RoboDK station: kr10 camera 070819 First 4 poses.rdk

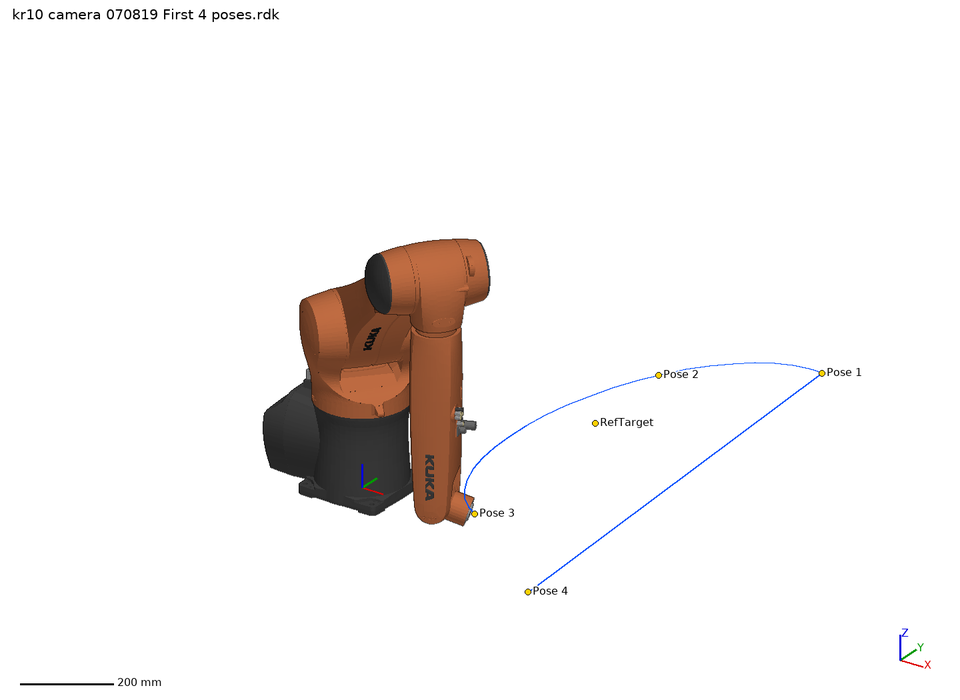
[picture v0: the station drawn from its stored meshes, robots at their saved joint values, targets as dots, program paths as lines]
Station kr10 camera 070819 First 4 poses. Poses are relative to the parent item; angles as X-Y-Z fixed-axis rotations.
  - frame KUKA KR 10 R1100 sixx Base at (0, 0, 0) mm
    - robot KUKA KR 10 R1100 sixx: 6 axes, payload 10 kg, reach 1101 mm, repeatability 0.03 mm, weight 54 kg
        modified DH rows (alpha deg, a mm, theta deg, d mm): 0, 0, 0, 400; -90, 25, 0, 0; 0, 560, -90, 0; -90, 35, 0, 515; 90, 0, 0, 0; -90, 0, 180, 80
        joint limits [-170, -190, -120, -185, -120, -350] to [170, 45, 156, 185, 120, 350]; home [0, -90, 90, 0, 0, 0]; saved at [37.108, -35.584, 126.083, 60.338, -72.571, -20.944]
      - tool Tool 1, TCP at (0, 0, 10) mm
    - target RefTarget (Cartesian target) at (609.71, 0, 323.9) mm, rotated rx 0 ry 90 rz 0 deg; joints [0, -49.182, 128.637, 0, -79.455, 0] of KUKA KR 10 R1100 sixx
    - target Pose 1 (Cartesian target) at (890.41, 444.52, 344) mm, rotated rx 147.73 ry 55.2 rz 49.99 deg; joints [-30.347, -18.532, 44.083, -131.002, -102.702, 30.664] of KUKA KR 10 R1100 sixx
    - target Pose 2 (Cartesian target) at (482.84, 415.27, 236.13) mm, rotated rx 133.49 ry 60.14 rz 73.16 deg; joints [-48.087, -38.36, 110.837, -109.682, -75.131, -5.051] of KUKA KR 10 R1100 sixx
    - target Pose 3 (Cartesian target) at (486.19, -274.25, 183.25) mm, rotated rx 131.13 ry 62.51 rz 151.14 deg; joints [37.108, -35.584, 126.083, 60.338, -72.571, -20.944] of KUKA KR 10 R1100 sixx
    - target Pose 4 (Cartesian target) at (798.41, -520.76, 183.47) mm, rotated rx 131.73 ry 63.14 rz -155.42 deg; joints [37.836, -12.412, 53.184, 118.846, -95.525, -64.778] of KUKA KR 10 R1100 sixx
  - Python program MoveL_Test_Make_Cube_Program (listed below)
  - program Prog2 (5 instructions, listed below)
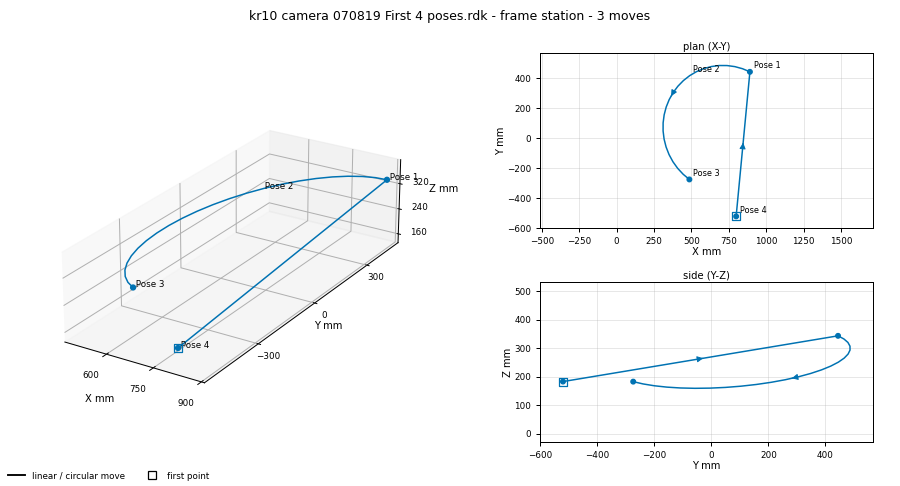
[picture p0: tool path of kr10 camera 070819 First 4 poses.rdk in frame station, 3 of 3 moves have a stored position in this frame; points joined in program order, loops and branches not executed]

--- Python program MoveL_Test_Make_Cube_Program ---
# This program shows how to use MoveL_Test to make sure that the robot can make a linear movement.
# This macro creates a cube of targets to follow by the robot
from robolink import *    # API to communicate with RoboDK
from robodk import *      # basic matrix operations
from random import uniform # to randomly calculate rz (rotation around the Z axis)

#Start the RoboDK API
RDK = Robolink()

# Run on robot: Force the program to run on the connected robot (same behavior as right clicking the program, then, selecting "Run on Robot")
# RDK.setRunMode(RUNMODE_RUN_ROBOT)

# Get the only robot in the station
robot = RDK.Item('', ITEM_TYPE_ROBOT)

# Get the target reference RefTarget
target_ref = RDK.Item('RefTarget')
# Get the reference position (pose=4x4 matrix of the target with respect to the reference frame)
pose_ref = target_ref.Pose()
startpoint = target_ref.Joints()
config_ref = robot.JointsConfig(startpoint)
tool_pose = robot.Childs()[0].PoseTool()

# Retrieve the degrees of freedom or axes (num_dofs = 6 for a 6 axis robot)
num_dofs = len(robot.JointsHome().list())

# Get the reference frame of the target reference
ref_frame = target_ref.Parent()

def config_equal(config1, config2):
    if config1[0] != config2[0] or config1[1] != config2[1] or config1[2] != config2[2]:
        return False
    return True


# Create a new program
prog = RDK.AddProgram('AutoCreated')

# This should make program generation slightly faster
#prog.ShowInstructions(False)

# Start creating the program or moving the robot:
program_or_robot = prog
program_or_robot.setPoseTool(tool_pose)

program_or_robot.MoveJ(target_ref)
lastjoints = startpoint
rz = 0
ntargets = 0
for tz in range(-100, 101, 100):
    for ty in range(0, 401, 200):
        for tx in range(100, -5001, -250):
            ntargets = ntargets + 1
            # calculate a random rotation around the Z axis of the tool
            #rz = uniform(-20*pi/180, 20*pi/180)

            # Calculate the position of the new target: translate with respect to the robot base and rotate around the tool
            newtarget_pose = transl(tx,ty,tz)*pose_ref*rotz(rz)

            # First, make sure the target is reachable:
            newtarget_joints = robot.SolveIK(newtarget_pose, lastjoints, tool_pose)
            if len(newtarget_joints.tolist()) < num_dofs:
                print('...target not reachable!! Skipping target')
                continue

            # Create a new target:
            newtarget_name = 'Auto T%.0f,%.0f,%.0f Rz=%.1f' % (tx,ty,tz,rz)
            print('Creating target %i: %s' % (ntargets, newtarget_name))
            newtarget = RDK.AddTarget(newtarget_name, ref_frame, robot)

            # At this point, the target is reachable.
            # We have to check if we can do a linear move or not. We have 2 methods:
            can_move_linear = True

            # ------------------------------
            # Validation method 1: check the joints at the destination target
            # and make sure we have the same configuration
            # A quick way to validate (it may not be perfect if robot joints can move more than 1 turn)
            # To improve this method we would have to check configurations on all possible solutions
            # from the inverse kinematics, using SolveIK_All()
            if False:
                target_joints_config = robot.JointsConfig(newtarget_joints)
                if not config_equal(config_ref, target_joints_config):
                    # We can't do a linear movement
                    can_move_linear = False
                    print("Warning! configuration is not the same as the reference target! Linear move will not be possible")

                    # update the reference configuration to the new one
                    config_ref = target_joints_config
            # -------------------------------



            # -------------------------------
            # Validation method 2: use the robot.MoveL_Test option to check if the robot can make a linear movement
            # This method is more robust and should provide a 100% accurate result but it may take more time
            # robot.MoveL_Test can also take collisions into account if collision checking is activated
            issues = robot.MoveL_Test(lastjoints, newtarget_pose)
            can_move_linear = (issues == 0)
            # We can retrieve the final joint position by retrieving the robot joints
            if can_move_linear:
                newtarget_joints = robot.Joints()

            # ---------------------------------

            if can_move_linear:
                # All good, we don't need to modify the target.
                # However, we could set the joints in the target as this may allow us to retrieve the robot configuration if we ever need it
                newtarget.setAsCartesianTarget() # default behavior
                newtarget.setJoints(newtarget_joints)
                # It is important to have setPose after setJoints as it may recalculate the joints to match the target
                newtarget.setPose(newtarget_pose)

                # Add the linear movement
                program_or_robot.MoveL(newtarget)

            else:
                print(newtarget_joints)
                # Make sure we have a joint target and a joint movement
                newtarget.setAsJointTarget() # default behavior

                # Setting the pose for a joint target is not important unless we want to retrieve the pose later
                # or we want to use the Cartesian coordinates for post processing
                newtarget.setPose(newtarget_pose)

                # Make sure we set the joints after the pose for a joint taget as it may recalculate the pose
                newtarget.setJoints(newtarget_joints)

                # Add the joint movement
                program_or_robot.MoveJ(newtarget)


            # Remember the joint poisition of the last movement
            lastjoints = newtarget_joints

# Showing the instructions at the end is faster:
prog.ShowInstructions(True)

# Hiding the targets is cleaner and more difficult to accidentaly move a target
#prog.ShowTargets(False)

print('Program done with %i targets' % ntargets)

--- program Prog2 (robot KUKA KR 10 R1100 sixx) ---
  Set Ref.: KUKA KR 10 R1100 sixx Base
  Set Tool: Tool 1
  MoveJ (Pose 4)
  MoveL (Pose 1)
  MoveC (Pose 2, Pose 3)
